ABB RobotStudio station: hanoi_v1vegleges.rspag

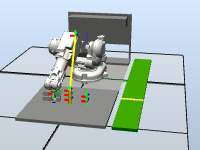
--- station ---
Station Solution3 (saved by RobotStudio format 3)
Controller IRB_140T_6kg_0.81m
  mechanical unit ROB_1: IRB140T_6_81_C_02, 6 joints, base frame (0, 0, 0) mm
Layout (positions relative to the parent item):
  - IRB140T_6_81_C_02 [mechanism, from Robots\IRB140T_6_81_C_G_02.rslib] at (0, 0, 0) mm; joint values [-0.2136, 1.3185, -0.6101, 0, 0.8624, -0.2136] (rad or m)
  - Henger1 [part] at (700, 0, 115.1) mm
  - Poz1 [part] at (-100, 50, 0.1) mm
  - Poz3 [part] at (-100, -50, 0.1) mm
  - SmatMefogo [smart component] at (691.11, -149.92, 129.64) mm, rotated rx 180 ry 0 rz -180 deg
      signals: DI Megfog, DI Elenged
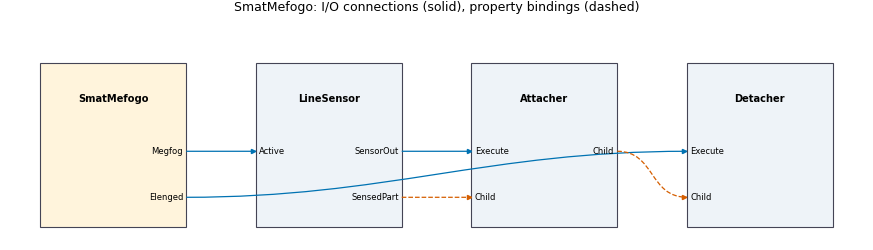
      connections:
        SmatMefogo.Megfog -> LineSensor.Active
        SmatMefogo.Elenged -> Detacher.Execute
        LineSensor.SensorOut -> Attacher.Execute
        LineSensor.SensedPart => Attacher.Child
        Attacher.Child => Detacher.Child
    - Megfogo [mechanism, from Libraries\Megfogo.rslib] at (0, 0, 0) mm, rotated rx 0 ry 0 rz -90 deg; joint values [0] (rad or m)
    - MegfogoTool [mechanism] at (0, 0, 0) mm
        TCP MyNewTool at (-15, 0, 70) mm, rotated rx -90 ry 0 rz -90 deg
        links: Dummy
    - LineSensor [smart component, from Components\LineSensor.rslib]
        properties: Start=[-0.0125 0.018 0.07]; End=[-0.0125 -0.019 0.07]; Radius=0.01; SensedPart=Henger1; SensedPoint=[0.700004211425781 0.0176903648376465 0.0605688705444336]
      - _sensorPart_ [part]
    - Attacher [smart component, from Components\Attacher.rslib]
        properties: Parent=Megfogo; Flange=0; Child=Henger1; Mount=false; Offset=[0 0 0]; Orientation=[0 0 0]
    - Detacher [smart component, from Components\Detacher.rslib]
        properties: Child=Henger1; KeepPosition=true
  - SmartFSzalag [smart component] at (24.45, 0, 0) mm
      signals: DI Activate, DO SzalagErzekel
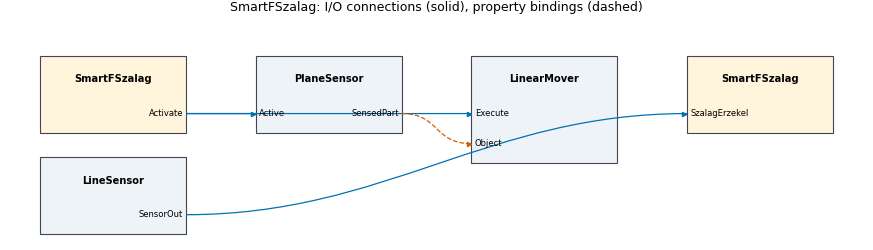
      connections:
        SmartFSzalag.Activate -> LinearMover.Execute
        SmartFSzalag.Activate -> PlaneSensor.Active
        LineSensor.SensorOut -> SmartFSzalag.SzalagErzekel
        PlaneSensor.SensedPart => LinearMover.Object
    - LinearMover [smart component, from Components\LinearMover.rslib]
        properties: Object=(none); Direction=[1 0 0]; Speed=0.1; Reference=Global; ReferenceObject=(none)
    - PlaneSensor [smart component, from Components\PlaneSensor.rslib]
        properties: Origin=[-0.7 0.425 0.027]; Axis1=[1.725 0 0]; Axis2=[0 0.2 0]; SensedPart=(none)
      - _sensorPart_ [part]
    - FutoSzalag [part] at (-700, 425, 0) mm
    - LineSensor [smart component, from Components\LineSensor.rslib]
        properties: Start=[0.525 0.625 0.045]; End=[0.525 0.425 0.045]; Radius=0.005; SensedPart=Henger1; SensedPoint=[0.525 0.497133544921875 0.045]
      - _sensorPart_ [part]
  - Poz2 [part] at (-100, -100, 0.1) mm
  - Asztal [part]
  - Henger2 [part] at (700, 0, 70.1) mm
  - Henger3 [part] at (700, 0, 25.1) mm
Attachment: SmatMefogo is attached to IRB140T_6_81_C_02 / Link6
EventTableEntry 959: Group=, Trigger=DO10_1 960, Actions=[EventTableActionMechanicalPose 961], Comment=, ActivationMode=2, Cyclic=false
EventTableTriggerIO 960: IOValue=[1], IRC5Controller=? -1, Operator=0, SignalSource=IRB_140T_6kg_0.81m 463
EventTableActionMechanicalPose 961: VirtualSignal=, Mechanism=Megfogo 970, ToPoseName=Elenged, VirtualSignalValue=[1]
EventTableEntry 988: Group=, Trigger=DO10_2 989, Actions=[EventTableActionMechanicalPose 990], Comment=, ActivationMode=2, Cyclic=false
EventTableTriggerIO 989: IOValue=[1], IRC5Controller=? -1, Operator=0, SignalSource=IRB_140T_6kg_0.81m 463
EventTableActionMechanicalPose 990: VirtualSignal=, Mechanism=Megfogo 970, ToPoseName=Megfog, VirtualSignalValue=[1]
Collision set CollisionSet_1: Henger1, Henger2, Henger3 against Asztal, near miss 0.005 m
Collision set CollisionSet_2: Henger1 against Henger2, near miss 0.005 m
Collision set CollisionSet_3: Henger2 against Henger3, near miss 0.005 m
Collision set CollisionSet_4: Henger1 against Henger3, near miss 0.005 m
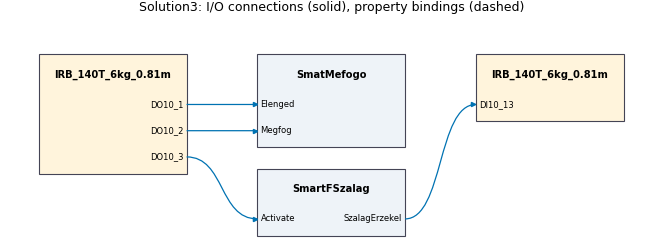
Station logic (signal -> signal, property => property):
  IRB_140T_6kg_0.81m.DO10_1 -> SmatMefogo.Elenged
  IRB_140T_6kg_0.81m.DO10_2 -> SmatMefogo.Megfog
  IRB_140T_6kg_0.81m.DO10_3 -> SmartFSzalag.Activate
  SmartFSzalag.SzalagErzekel -> IRB_140T_6kg_0.81m.DI10_13

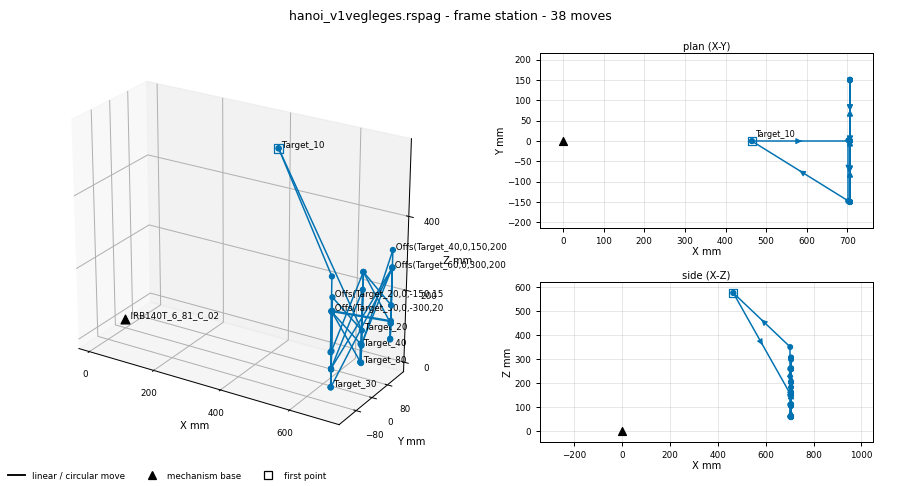
[picture p0: tool path of hanoi_v1vegleges.rspag in frame station, 38 of 38 moves have a stored position in this frame; points joined in program order, loops and branches not executed]
--- Backups/IRB_140T_6kg_0.81m/RAPID/TASK1/PROGMOD/CalibData.mod ---
MODULE CalibData
	PERS tooldata MegfogoTool:=[TRUE,[[-15,0,70],[0.5,-0.5,0.5,-0.5]],[1,[0,0,1],[1,0,0,0],0,0,0]];
	PERS tooldata MyNewTool:=[TRUE,[[-15,0,70],[0.5,-0.5,0.5,-0.5]],[1,[0,0,1],[1,0,0,0],0,0,0]];
ENDMODULE

--- Backups/IRB_140T_6kg_0.81m/RAPID/TASK1/PROGMOD/Module1.mod ---
MODULE Module1
	CONST robtarget Target_10:=[[465.000042379,0,577.000004709],[0.499999922,0.500000078,-0.500000078,-0.499999922],[0,0,0,0],[9E9,9E9,9E9,9E9,9E9,9E9]];
	CONST robtarget Target_20:=[[706.29148314,0,149.027341333],[0.499999676,0.500000324,-0.500000324,-0.499999676],[0,0,0,0],[9E9,9E9,9E9,9E9,9E9,9E9]];
	CONST robtarget Target_30:=[[706.081910176,-150.06169164,58.935787972],[0.499999074,0.500000376,-0.500001266,-0.499999284],[-1,0,-1,0],[9E9,9E9,9E9,9E9,9E9,9E9]];
	CONST robtarget Target_40:=[[706.10501062,0.373088974,107.63005266],[0.499999278,0.500000547,-0.5000011,-0.499999074],[0,-1,0,0],[9E9,9E9,9E9,9E9,9E9,9E9]];
	CONST robtarget Target_50:=[[706.105462967,150.590701376,63.243395269],[0.499998785,0.500001362,-0.500001362,-0.499998491],[0,-1,0,0],[9E9,9E9,9E9,9E9,9E9,9E9]];
	CONST robtarget Target_60:=[[706.105265073,-149.380670844,58.351871655],[0.499998898,0.500001449,-0.500000817,-0.499998837],[-1,0,-1,0],[9E9,9E9,9E9,9E9,9E9,9E9]];
	CONST robtarget Target_70:=[[706.105123246,150.986861049,105.99976202],[0.499999269,0.50000123,-0.500000379,-0.499999122],[0,-1,0,0],[9E9,9E9,9E9,9E9,9E9,9E9]];
	CONST robtarget Target_80:=[[706.105211733,-0.001957075,59.739782525],[0.499999308,0.500001348,-0.500000329,-0.499999015],[-1,0,-1,0],[9E9,9E9,9E9,9E9,9E9,9E9]];
	CONST robtarget Target_90:=[[706.105644252,-149.916156259,59.643989983],[0.499998898,0.500001448,-0.500000817,-0.499998836],[-1,0,-1,0],[9E9,9E9,9E9,9E9,9E9,9E9]];
	CONST robtarget Target_100:=[[706.105446407,150.724824762,105.747464592],[0.499999252,0.500001247,-0.500000391,-0.49999911],[0,-1,0,0],[9E9,9E9,9E9,9E9,9E9,9E9]];
	CONST robtarget Target_110:=[[706.105105603,0.34774307,60.713177425],[0.499999579,0.500001047,-0.500000093,-0.499999281],[0,0,0,0],[9E9,9E9,9E9,9E9,9E9,9E9]];
	CONST robtarget Target_120:=[[706.105457934,150.459882019,61.116532435],[0.499999256,0.500001251,-0.500000388,-0.499999106],[0,-1,0,0],[9E9,9E9,9E9,9E9,9E9,9E9]];
	CONST robtarget Target_130:=[[706.105526904,-149.232431087,106.444105119],[0.499999103,0.500001278,-0.500000469,-0.49999915],[-1,0,-1,0],[9E9,9E9,9E9,9E9,9E9,9E9]];
	CONST robtarget Target_140:=[[702.50422999,2.109371519,60.568872111],[0.49999931,0.500000843,-0.500000326,-0.499999521],[0,0,0,0],[9E9,9E9,9E9,9E9,9E9,9E9]];
	CONST robtarget Target_150:=[[702.504410618,-147.464295053,151.335460389],[0.49999882,0.500001096,-0.500000743,-0.499999341],[-1,0,-1,0],[9E9,9E9,9E9,9E9,9E9,9E9]];
    PROC Megfog()
        PulseDO DO10_2;
        WaitTime 1;
    ENDPROC
    PROC Elenged()
        PulseDO DO10_1;
        WaitTime 1;
    ENDPROC
	PROC Path_10()
	    MoveJ Target_10,v100,fine,MegfogoTool\WObj:=wobj0;
	    MoveL Target_20,v100,fine,MegfogoTool\WObj:=wobj0;
        Megfog;
        MoveL Offs(Target_20,0,-150,150),v100,fine,MegfogoTool\WObj:=wobj0;
	    MoveL Target_30,v100,fine,MegfogoTool\WObj:=wobj0;
        Elenged;
        MoveL Offs(Target_30,0,0,50),v100,fine,MegfogoTool\WObj:=wobj0;
        MoveL Offs(Target_30,0,150,200),v100,fine,MegfogoTool\WObj:=wobj0;
	    MoveL Target_40,v100,fine,MegfogoTool\WObj:=wobj0;
        Megfog;
        MoveL Offs(Target_40,0,150,200),v100,fine,MegfogoTool\WObj:=wobj0;
	    MoveL Target_50,v100,fine,MegfogoTool\WObj:=wobj0;
        Elenged;
        MoveL Offs(Target_50,0,0,50),v100,fine,MegfogoTool\WObj:=wobj0;
        MoveL Offs(Target_50,0,-300,200),v100,fine,MegfogoTool\WObj:=wobj0;
	    MoveL Target_60,v100,fine,MegfogoTool\WObj:=wobj0;
	    Megfog;
        MoveL Offs(Target_60,0,300,200),v100,fine,MegfogoTool\WObj:=wobj0;
        MoveL Target_70,v100,fine,MegfogoTool\WObj:=wobj0;
	    Elenged;
        MoveL Offs(Target_70,0,0,50),v100,fine,MegfogoTool\WObj:=wobj0;
        MoveL Offs(Target_70,0,-150,200),v100,fine,MegfogoTool\WObj:=wobj0;
        MoveL Target_80,v100,fine,MegfogoTool\WObj:=wobj0;
	    Megfog;
        MoveL Offs(Target_80,0,-150,200),v100,fine,MegfogoTool\WObj:=wobj0;
        MoveL Target_90,v100,fine,MegfogoTool\WObj:=wobj0;
	    Elenged;
        MoveL Offs(Target_90,0,0,50),v100,fine,MegfogoTool\WObj:=wobj0;
        MoveL Offs(Target_90,0,300,200),v100,fine,MegfogoTool\WObj:=wobj0;
        MoveL Target_100,v100,fine,MegfogoTool\WObj:=wobj0;
	    Megfog;
        MoveL Offs(Target_100,0,-150,200),v100,fine,MegfogoTool\WObj:=wobj0;
        MoveL Target_110,v100,fine,MegfogoTool\WObj:=wobj0;
	    Elenged;
        MoveL Offs(Target_110,0,0,50),v100,fine,MegfogoTool\WObj:=wobj0;
        MoveL Offs(Target_110,0,150,200),v100,fine,MegfogoTool\WObj:=wobj0;
        MoveL Target_120,v100,fine,MegfogoTool\WObj:=wobj0;
	    Megfog;
        MoveL Offs(Target_120,0,0,50),v100,fine,MegfogoTool\WObj:=wobj0;
        MoveL Offs(Target_120,0,-300,200),v100,fine,MegfogoTool\WObj:=wobj0;
        MoveL Target_130,v100,fine,MegfogoTool\WObj:=wobj0;
	    Elenged;
        MoveL Offs(Target_130,0,0,50),v100,fine,MegfogoTool\WObj:=wobj0;
        MoveL Offs(Target_130,0,150,200),v100,fine,MegfogoTool\WObj:=wobj0;
        MoveL Target_140,v100,fine,MegfogoTool\WObj:=wobj0;
	    Megfog;
        MoveL Offs(Target_140,0,0,50),v100,fine,MegfogoTool\WObj:=wobj0;
        MoveL Offs(Target_140,0,-150,200),v100,fine,MegfogoTool\WObj:=wobj0;
        MoveL Target_150,v100,fine,MegfogoTool\WObj:=wobj0;
        Elenged;
        MoveL Offs(Target_150,0,0,200),v100,fine,MegfogoTool\WObj:=wobj0;
        MoveL Target_10,v100,fine,MegfogoTool\WObj:=wobj0;
	ENDPROC
    PROC main()
    Path_10;
    ENDPROC
ENDMODULE

--- Backups/IRB_140T_6kg_0.81m/RAPID/TASK1/PROGMOD/RsTempModule.mod ---
MODULE RsTempModule
	PERS wobjdata wobj02:=[FALSE,TRUE,"",[[0,0,0],[1,0,0,0]],[[0,0,0],[1,0,0,0]]];
	PERS tooldata MegfogoTool1:=[TRUE,[[-15,0,70],[0.5,-0.5,0.5,-0.5]],[1,[0,0,1],[1,0,0,0],0,0,0]];
PROC RsTempPath()
ENDPROC

ENDMODULE

--- Backups/IRB_140T_6kg_0.81m/RAPID/TASK1/SYSMOD/LINKEDM.sys ---
%%%
  VERSION:1
  LANGUAGE:ENGLISH
%%%

MODULE LINKEDM (SYSMODULE)

! FOLLOWER
!     Name of electronically linked follower axis used by operator at teach pendent.
      PERS string l_f_axis_name{5}       :=  ["",  "", "", "", ""];

!     Name of the mechanical unit for follower axis.
      PERS string l_f_mecunt_n{5}  :=  ["", "", "", "", ""];

!     Linked follower axis number in the mechanical unit (first axis in mech. unit is number 1).
      PERS num l_f_axis_no{5}      :=  [0,          0,   0,  0,  0];

! MASTER
!     Name of the mechanical unit for linked master axis.
      PERS string l_m_mecunt_n{5} :=  ["", "", "", "", ""];

!     Linked master axis number in the mechanical unit (first axis in mech. unit is number 1).
!     See axis number table in documentation for different master mechanical units.
      PERS num l_m_axis_no{5}     :=  [0,  0,  0,  0,  0];

! POSITION OFFSET
!     The increase of the allowed offset position between the master and follower
!     positions, used when starting AUTO mode. As soon as the offset is decreased
!     the old configurated parameter is used.
!     Example: 3 => the configurated value of allowed offset is increased 3 times.
      PERS num offset_ratio{5}       :=  [10,  10,   10,  10,  10];

! SPEED RATIO
!     Speed_ratio used in AUTO and JOG modes [ very_slow   slow    normal    fast]
!     Value 1 = max allowed manual speed.
      CONST num speed_ratio {20}      := [0.01, 0.01, 0.01, 0.01, 0.01,
                                          0.05, 0.05, 0.05, 0.05, 0.05,
                                          0.20, 0.20, 0.20, 0.20, 0.20,
                                          1.00, 1.00, 1.00, 1.00, 1.00];

! STEP SIZE
!     Displacement position used in JOG mode for each activation of positive or
!     negative movement.                  [very_short    short   normal   long]
!     Unit degees or meter.
      CONST num displacement {20}     := [0.001, 0.001, 0.001, 0.001, 0.001,
                                          0.005, 0.005, 0.005, 0.005, 0.005,
                                          0.020, 0.020, 0.020, 0.020, 0.020,
                                          0.100, 0.100, 0.100, 0.100, 0.100];


!-------------------------------------------------------------
 PROC Linked_m ()
      Linked_m_exe ;
 ENDPROC
ENDMODULE

--- Backups/IRB_140T_6kg_0.81m/SYSPAR/EIO.cfg ---
EIO:CFG_1.0:6:0::
#
EIO_SIGNAL:

      -Name "DO10_1" -SignalType "DO" -Access "All"

      -Name "DO10_2" -SignalType "DO" -Access "All"

      -Name "DO10_3" -SignalType "DO" -Access "All"

      -Name "DI10_13" -SignalType "DI" -Access "All"
